FUNCTION ARCSEC_TO_RAD : LREAL
VAR_INPUT
    arcsec : LREAL;
END_VAR
VAR
END_VAR

ARCSEC_TO_RAD := DEG_TO_RAD(ARCSEC_TO_DEG(arcsec));

END_FUNCTION

(* stored: Version 1.1.0.1, ProductVersion 3.1.4019.2
   POU ARCSEC_TO_RAD: Id {00eb3aec-c58d-4f39-becf-cbe5f70d3551}, SpecialFunc None *)
